FUNCTION_BLOCK AxesIO EXTENDS SM_AxesIO
VAR_INPUT
END_VAR
VAR_OUTPUT
END_VAR
VAR
    _testVar : BOOL; // without any variable, the superclass attributes are not visible in the UA address space
END_VAR

SUPER^();

// do stuff

//SUPER^();

END_FUNCTION_BLOCK

(* stored: Version 1.1.0.1, ProductVersion 3.1.4018.5
   POU AxesIO: Id {ed130642-6a7b-47c8-adb8-b940941127ae}, SpecialFunc None *)
